TYPE "POWDER FEEDER HMI ACTIONS"
// stored: IsFailsafeCompliant false
   STRUCT
      SWITCH_ON_HEATER_LINE_1 : Bool;   // SWITCH ON HEATER LINE 1 HMI REQUEST
      SWITCH_OFF_HEATER_LINE_1 : Bool;   // SWITCH OFF HEATER LINE 1 HMI REQUEST
      SWITCHED_ON_HEATER_LINE_1 : Bool;   // SWITCHED ON HEATER LINE 1 HMI STATUS
      SWITCHED_OFF_HEATER_LINE_1 : Bool;   // SWITCHED OFF HEATER LINE 1 HMI STATUS
      SWITCH_ON_HEATER_LINE_2 : Bool;   // SWITCH ON HEATER LINE 2 HMI REQUEST
      SWITCH_OFF_HEATER_LINE_2 : Bool;   // SWITCH OFF HEATER LINE 2 HMI REQUEST
      SWITCHED_ON_HEATER_LINE_2 : Bool;   // SWITCHED ON HEATER LINE 2 HMI STATUS
      SWITCHED_OFF_HEATER_LINE_2 : Bool;   // SWITCHED OFF HEATER LINE 2 HMI STATUS
      SWITCH_ON_HOOPER_LINE_1 : Bool;   // SWITCH ON HOOPER LINE 1 HMI REQUEST
      SWITCH_OFF_HOOPER_LINE_1 : Bool;   // SWITCH OFF HOOPER LINE 1 HMI REQUEST
      SWITCHED_ON_HOOPER_LINE_1 : Bool;   // SWITCHED ON HOOPER LINE 1 HMI STATUS
      SWITCHED_OFF_HOOPER_LINE_1 : Bool;   // SWITCHED OFF HOOPER LINE 1 HMI STATUS
      SWITCH_ON_HOOPER_LINE_2 : Bool;   // SWITCH ON HOOPER LINE 2 HMI REQUEST
      SWITCH_OFF_HOOPER_LINE_2 : Bool;   // SWITCH OFF HOOPER LINE 2 HMI REQUEST
      SWITCHED_ON_HOOPER_LINE_2 : Bool;   // SWITCHED ON HOOPER LINE 2 HMI STATUS
      SWITCHED_OFF_HOOPER_LINE_2 : Bool;   // SWITCHED OFF HOOPER LINE 2 HMI STATUS
      SELECT_ARGON_GAS : Bool;   // SELECT ARGON GAS HMI REQUEST
      SELECT_NITROGEN_GAS : Bool;   // SELECT NITROGEN GAS HMI REQUEST
      SELECT_HELIUM_GAS : Bool;   // SELECT HELIUM GAS HMI REQUEST
      SELECT_ARGON30_GAS : Bool;   // SELECT ARGON30 GAS HMI REQUEST
      SELECTED_ARGON_GAS : Bool;   // SELECTED ARGON GAS HMI STATUS
      SELECTED_NITROGEN_GAS : Bool;   // SELECTED NITROGEN GAS HMI STATUS
      SELECTED_HELIUM_GAS : Bool;   // SELECTED HELIJM GAS HMI STATUS
      SELECTED_ARGON30_GAS : Bool;   // SELECTED ARGON30 GAS HMI STATUS
      SELECT_METRIC_UNITS : Bool;   // SELECT METRIC UNITS HMI REQUEST
      SELECT_IMPERIAL_UNITS : Bool;   // SELECT IMPERIAL UNITS HMI REQUEST
      SELECTED_METRIC_UNITS : Bool;   // SELECTED METRIC UNITS HMI STATUS
      SELECTED_IMPERIAL_UNITS : Bool;   // SELECTED IMPERIAL UNITS HMI STATUS
   END_STRUCT;
END_TYPE

TYPE "POWDER FEEDER HMI OFFSETS ALARMS WARNINGS"
// stored: IsFailsafeCompliant false
   STRUCT
      CarrierGasNominalLine1_Max_Alarm : Real;
      CarrierGasNominalLine2_Max_Alarm : Real;
      DiskSpeedNominalLine1_Max_Alarm : Real;
      DiskSpeedNominalLine2_Max_Alarm : Real;
      StirrerSpeedNominalLine1_Max_Alarm : Real;
      StirrerSpeedNominalLine2_Max_Alarm : Real;
      HopperTempNominalLine1_Max_Alarm : Real;
      HopperTempNominalLine2_Max_Alarm : Real;
      CarrierGasNominalLine1_Min_Alarm : Real;
      CarrierGasNominalLine2_Min_Alarm : Real;
      DiskSpeedNominalLine1_Min_Alarm : Real;
      DiskSpeedNominalLine2_Min_Alarm : Real;
      StirrerSpeedNominalLine1_Min_Alarm : Real;
      StirrerSpeedNominalLine2_Min_Alarm : Real;
      CarrierGasNominalLine1_Max_Warning : Real;
      CarrierGasNominalLine2_Max_Warning : Real;
      DiskSpeedNominalLine1_Max_Warning : Real;
      DiskSpeedNominalLine2_Max_Warning : Real;
      StirrerSpeedNominalLine1_Max_Warning : Real;
      StirrerSpeedNominalLine2_Max_Warning : Real;
      CarrierGasNominalLine1_Min_Warning : Real;
      CarrierGasNominalLine2_Min_Warning : Real;
      DiskSpeedNominalLine1_Min_Warning : Real;
      DiskSpeedNominalLine2_Min_Warning : Real;
      StirrerSpeedNominalLine1_Min_Warning : Real;
      StirrerSpeedNominalLine2_Min_Warning : Real;
      Spare26 : Real;
      Spare27 : Real;
      Spare28 : Real;
      Spare29 : Real;
      Spare30 : Real;
   END_STRUCT;
END_TYPE

TYPE "POWDER FEEDER HMI VALUES SETPOINTS"
// stored: IsFailsafeCompliant false
   STRUCT
      CarrierGasNominalLine1 : Real;
      CarrierGasNominalLine2 : Real;
      DiskSpeedNominalLine1 : Real;
      DiskSpeedNominalLine2 : Real;
      StirrerSpeedNominalLine1 : Real;
      StirrerSpeedNominalLine2 : Real;
      HopperTempNominalLine1 : Real;
      HopperTempNominalLine2 : Real;
      Spare8 : Real;
      Spare9 : Real;
      Spare10 : Real;
      Spare11 : Real;
      Spare12 : Real;
      Spare13 : Real;
      Spare14 : Real;
      Spare15 : Real;
   END_STRUCT;
END_TYPE

TYPE "POWDER FEEDER HOPPER"
// stored: IsFailsafeCompliant false
   STRUCT
      START_GENERAL_CONDITIONS : Bool;   // START GENERAL CONDITIONS
      START_INITIAL_CONDITIONS_LINE_1 : Bool;   // START INITIAL CONDITIONS LINE 1
      START_MANUAL_REQUEST_LINE_1 : Bool;   // START MANUAL REQUEST LINE 1
      START_INITIAL_CONDITIONS_LINE_2 : Bool;   // START INITIAL CONDITIONS LINE 2
      START_MANUAL_REQUEST_LINE_2 : Bool;   // START MANUAL REQUEST LINE 2
      START_AUTO_REQUEST : Bool;   // START AUTO REQUEST
      START_GLOBAL_REQUEST_LINE_1 : Bool;   // START GLOBAL REQUEST LINE 1
      START_COMMAND_LINE_1 : Bool;   // START COMMAND LINE 1
      START_LINE_1 : Bool;   // START LINE 1
      FEEDBACK_ON_LINE_1 : Bool;   // FEEDBACK ON LINE 1
      START_GLOBAL_REQUEST_LINE_2 : Bool;   // START GLOBAL REQUEST LINE 2
      START_COMMAND_LINE_2 : Bool;   // START COMMAND LINE 2
      START_LINE_2 : Bool;   // START LINE 2
      FEEDBACK_ON_LINE_2 : Bool;   // FEEDBACK ON LINE 2
      STOP_GENERAL_CONDITIONS : Bool;   // STOP GENERAL CONDITIONS
      STOP_INITIAL_CONDITIONS_LINE_1 : Bool;   // STOP INITIAL CONDITIONS LINE 1
      STOP_MANUAL_REQUEST_LINE_1 : Bool;   // STOP MANUAL REQUEST LINE 1
      STOP_INITIAL_CONDITIONS_LINE_2 : Bool;   // STOP INITIAL CONDITIONS LINE 2
      STOP_MANUAL_REQUEST_LINE_2 : Bool;   // STOP MANUAL REQUEST LINE 2
      STOP_AUTO_REQUEST : Bool;   // STOP AUTO REQUEST
      STOP_GLOBAL_REQUEST_LINE_1 : Bool;   // STOP GLOBAL REQUEST LINE 1
      STOP_COMMAND_LINE_1 : Bool;   // STOP COMMAND LINE 1
      STOP_LINE_1 : Bool;   // STOP LINE 1
      FEEDBACK_OFF_LINE_1 : Bool;   // FEEDBACK OFF LINE 1
      STOP_GLOBAL_REQUEST_LINE_2 : Bool;   // STOP GLOBAL REQUEST LINE 2
      STOP_COMMAND_LINE_2 : Bool;   // STOP COMMAND LINE 2
      STOP_LINE_2 : Bool;   // STOP LINE 2
      FEEDBACK_OFF_LINE_2 : Bool;   // FEEDBACK OFF LINE 2
      START_GENERAL_CONDITIONS_HELP : Bool;   // START GENERAL CONDITIONS HELP
      START_INITIAL_CONDITIONS_HELP : Bool;   // START INITIAL CONDITIONS HELP
      STOP_GENERAL_CONDITIONS_HELP : Bool;   // STOP GENERAL CONDITIONS HELP
      STOP_INITIAL_CONDITIONS_HELP : Bool;   // STOP INITIAL CONDITIONS HELP
      FAULT : Bool;   // FAULT
   END_STRUCT;
END_TYPE

TYPE "POWDER FEEDER PLC AUXILIAR"
// stored: IsFailsafeCompliant false
   STRUCT
      o_fCarrierGasSelect : Bool;   // 0 = Argon Selected, 1 = Nitrogen Selected / 1 = Argon, 2 = Nitrogen, 3 = Helium, 4 = Argon30
      o_fUnitSelect : Bool;   // 0 = Metric Units, 1 = SI
      i_fCarrierGasSelected_Line1 : Bool;   // 0 = Argon Selected, 1 = Nitrogen Selected / 1 = Argon, 2 = Nitrogen, 3 = Helium, 4 = Argon30
      i_fCarrierGasSelected_Line2 : Bool;   // 0 = Argon Selected, 1 = Nitrogen Selected / 1 = Argon, 2 = Nitrogen, 3 = Helium, 4 = Argon30
      i_fCarrierGasSelectedAux : Bool;   // 1 = Argon, 2 = Nitrogen, 3 = Helium, 4 = Argon30
      i_fUnitSelected_Line1 : Bool;   // 0 = Metric Units, 1 = SI / 0 = Metric System, 1 = Imperial
      i_fUnitSelected_Line2 : Bool;   // 0 = Metric Units, 1 = SI / 0 = Metric System, 1 = Imperial
      i_fUnitSelectedAux : Bool;   // 0 = Metric System, 1 = Imperial
      o_rCarriergasNominal_Line1 : Real;   // Carrier Gas Setpoint [NLPM] (0..16 NLPM)
      o_rCarriergasNominal_Line2 : Real;   // Carrier Gas Setpoint [NLPM] (0..16 NLPM)
      o_rDiskSpeedNominal_Line1 : Real;   // Disk Speed Setpoint [%] (0..100 %)
      o_rDiskSpeedNominal_Line2 : Real;   // Disk Speed Setpoint [%] (0..100 %)
      o_rStirrerSpeedNominal_Line1 : Real;   // Stirrer Speed Setpoint [%] (30 - 100%)
      o_rStirrerSpeedNominal_Line2 : Real;   // Stirrer Speed Setpoint [%] (30 - 100%)
      o_rHopperTempNominal_Line1 : Real;   // Hopper Temperature Setpoint [°C] (n/a for Twin 150 R1.0)
      o_rHopperTempNominal_Line2 : Real;   // Hopper Temperature Setpoint [°C] (n/a for Twin 150 R1.0)
      o_rLLlimitCarriergas_Line1 : Real;   // Carrier Gas Flow LL Limit [NLPM] (Absolute Value)
      o_rLLlimitCarriergas_Line2 : Real;   // Carrier Gas Flow LL Limit [NLPM] (Absolute Value)
      o_rLLlimitDiskSpeedNominal_Line1 : Real;   // Disk Speed LL Limit [%] (Absolute Value)
      o_rLLlimitDiskSpeedNominal_Line2 : Real;   // Disk Speed LL Limit [%] (Absolute Value)
      o_rLLlimitStirrerSpeedNominal_Line1 : Real;   // Stirrer Speed LL Limit [%] (Absolute Value)
      o_rLLlimitStirrerSpeedNominal_Line2 : Real;   // Stirrer Speed LL Limit [%] (Absolute Value)
      o_rLlimitCarriergas_Line1 : Real;   // Carrier Gas L Limit [NLPM] (Absolute Value)
      o_rLlimitCarriergas_Line2 : Real;   // Carrier Gas L Limit [NLPM] (Absolute Value)
      o_rLlimitDiskSpeedNominal_Line1 : Real;   // Disk Speed L Limit [%] (Absolute Value)
      o_rLlimitDiskSpeedNominal_Line2 : Real;   // Disk Speed L Limit [%] (Absolute Value)
      o_rLlimitStirrerSpeedNominal_Line1 : Real;   // Stirrer Speed L Limit [%] (Absolute Value)
      o_rLlimitStirrerSpeedNominal_Line2 : Real;   // Stirrer Speed L Limit [%] (Absolute Value)
      o_rHlimitCarriergas_Line1 : Real;   // Carrier Gas H Limit [NLPM] (Absolute Value)
      o_rHlimitCarriergas_Line2 : Real;   // Carrier Gas H Limit [NLPM] (Absolute Value)
      o_rHlimitDiskSpeedNominal_Line1 : Real;   // Disk Speed H Limit [%] (Absolute Value)
      o_rHlimitDiskSpeedNominal_Line2 : Real;   // Disk Speed H Limit [%] (Absolute Value)
      o_rHlimitStirrerSpeedNominal_Line1 : Real;   // Stirrer Speed H Limit [%] (Absolute Value)
      o_rHlimitStirrerSpeedNominal_Line2 : Real;   // Stirrer Speed H Limit [%] (Absolute Value)
      o_rHHlimitCarriergas_Line1 : Real;   // Carrier Gas HH Limit [NLPM] (Absolute Value)
      o_rHHlimitCarriergas_Line2 : Real;   // Carrier Gas HH Limit [NLPM] (Absolute Value)
      o_rHHlimitDiskSpeedNominal_Line1 : Real;   // Disk Speed HH Limit [%] (Absolute Value)
      o_rHHlimitDiskSpeedNominal_Line2 : Real;   // Disk Speed HH Limit [%] (Absolute Value)
      o_rHHlimitStirrerSpeedNominal_Line1 : Real;   // Stirrer Speed HH Limit [%] (Absolute Value)
      o_rHHlimitStirrerSpeedNominal_Line2 : Real;   // Stirrer Speed HH Limit [%] (Absolute Value)
      o_rHHlimitHopperTempNominal_Line1 : Real;   // Hopper Temperature HH Limit (ºC), (Absolute Value, N/a For Twin 150 R1.0)
      o_rHHlimitHopperTempNominal_Line2 : Real;   // Hopper Temperature HH Limit (ºC), (Absolute Value, N/a For Twin 150 R1.0)
      i_rCarriergasActual_Line1 : Real;   // Actual Value Carriergas Flow (NLPM)
      i_rCarriergasActual_Line2 : Real;   // Actual Value Carriergas Flow (NLPM)
      i_rDiskActual_Line1 : Real;   // Actual Value Disk Speed (%)
      i_rDiskActual_Line2 : Real;   // Actual Value Disk Speed (%)
      i_rStirrerActual_Line1 : Real;   // Actual Value Stirrer Speed (%)
      i_rStirrerActual_Line2 : Real;   // Actual Value Stirrer Speed (%)
      i_rFeedrateActual_Line1 : Real;   // N/A For Twin 150
      i_rFeedrateActual_Line2 : Real;   // N/A For Twin 150
      i_rHopperTempActual_Line1 : Real;   // Actual Value Hopper Temperature (ºC)
      i_rHopperTempActual_Line2 : Real;   // Actual Value Hopper Temperature (ºC)
      i_rHopperPressureActual_Line1 : Real;   // Actual Value Hopper Pressure (Bar)
      i_rHopperPressureActual_Line2 : Real;   // Actual Value Hopper Pressure (Bar)
   END_STRUCT;
END_TYPE

TYPE "POWDER SWITCH"
// stored: IsFailsafeCompliant false
   STRUCT
      "Hopper 1 General Conditions" : Bool;   // Hopper 1 General Conditions
      "Hopper 1 Initial Conditions" : Bool;   // Hopper 1 Initial Conditions
      "Hopper 1 Manual Request" : Bool;   // Hopper 1 Manual Request
      "Hopper 1 Auto Request" : Bool;   // Hopper 1 Auto Request
      "Hopper 1 Global Request" : Bool;   // Hopper 1 Global Request
      "Hopper 1 Command" : Bool;   // Hopper 1 Command
      "Hopper 1" : Bool;   // Hopper 1
      "Feedback Hopper 1" : Bool;   // Feedback Hopper 1
      "Hopper 2 General Conditions" : Bool;   // Hopper 2 General Conditions
      "Hopper 2 Initial Conditions" : Bool;   // Hopper 2 Initial Conditions
      "Hopper 2 Manual Request" : Bool;   // Hopper 2 Manual Request
      "Hopper 2 Auto Request" : Bool;   // Hopper 2 Auto Request
      "Hopper 2 Global Request" : Bool;   // Hopper 2 Global Request
      "Hopper 2 Command" : Bool;   // Hopper 2 Command
      "Hopper 2" : Bool;   // Hopper 2
      "Feedback Hopper 2" : Bool;   // Feedback Hopper 2
      "Hopper 1 General Conditions Help" : Bool;   // Hopper 1 General Conditions Help
      "Hopper 1 Initial Conditions Help" : Bool;   // Hopper 1 Initial Conditions Help
      "Hopper 2 General Conditions Help" : Bool;   // Hopper 2 General Conditions Help
      "Hopper 2 Initial Conditions Help" : Bool;   // Hopper 2 Initial Conditions Help
   END_STRUCT;
END_TYPE

TYPE "LBP_typeAlarmMsgs"
TITLE = PLC-Error / Messages / PLC errores/avisos / PLC-Fehler / Meldungen
// User data type for block LBP_AlarmMessage [DB2] / Tipo de dato de usuario para bloque LBP_AlarmMessage [DB2] / Anwender-Datentyp für Baustein LBP_AlarmMessage [DB2]
// stored: IsFailsafeCompliant false
   STRUCT
      Chan : Array[1..10] of Struct   // Von Kanal 1..10 / From Channel 1..10 / Desde el canal 1..10
         FDD : Array[0..15] of Bool;   // Vorschub deaktivieren / Feed disable / Desactivar avance
         RID : Array[0..15] of Bool;   // Einlesen deaktivieren / Read-in disable / Desactivar lectura
         NCSD : Array[0..15] of Bool;   // NC Start deaktivieren / NC start disable / Desactivar Marcha CN
         FdStop_1 : Array[0..15] of Bool;   // Vorschub-Stopp GEO-Achse 1 / Feed stop GEOaxis 1 / Parada del avance eje geométrico 1
         FdStop_2 : Array[0..15] of Bool;   // Vorschub-Stopp GEO-Achse 2 / Feed stop GEOaxis 2 / Parada del avance eje geométrico 2
         FdStop_3 : Array[0..15] of Bool;   // Vorschub-Stopp GEO-Achse 3 / Feed stop GEOaxis 3 / Parada del avance eje geométrico 3
      END_STRUCT;
      Axis : Array[1..31] of Struct   // Von Achse 1..31 / From Axis 1..31 / Desde el eje 1..31
         FdStop : Array[0..15] of Bool;   // Vorschub-Stopp Achse/Spindel / Feed stop axis/spindle / Parada del avance eje/cabezal
      END_STRUCT;
      AddValUserA0 : Array[0..63] of Int;   // Zusätzlicher Wert für Alarme im Anwenderbereich 0 (700000..700063) / Additional value for alarms in the user area 0 (700000..700063) / Valor adicional para alarmas en el área de usuario 0 (700000..700063)
      ChanA : Array[1..10] of Struct   // Von Kanal 1..10 / From Channel 1..10 / Desde el canal 1..10
         FDD_5C00xx : Array[0..15] of Bool;   // Vorschub deaktivieren Alarm Nr. 5C0000..5C0015 / Feed disable Alarm no. 5C0000..5C0015 / Desactivar avance n.º alarma 5C0000..5C0015
         FDD_RID_5C01xx : Array[0..31] of Bool;   // Vorschub und Einlesen deaktivieren Alarm Nr. 5C0100..5C0131 / Feed and read-in disable Alarm no. 5C0100..5C0131 / Desactivar avance y lectura n.º alarma 5C0100..5C0131
         RID_5C02xx : Array[0..31] of Bool;   // Einlesen deaktivieren Alarm Nr. 5C0200..5C0231 / Read-in disable Alarm no. 5C0200..5C0231 / Desactivar lectura n.º alarma 5C0200..5C0231
         NCSD_5C03xx : Array[0..15] of Bool;   // NC Start deaktivieren Alarm Nr. 5C0300..5C0315 / NC start disable Alarm no. 5C0300..5C0315 / Desactivar Marcha CN n.º alarma 5C0300..5C0315
         FdStop_1_5C11xx : Array[0..15] of Bool;   // Vorschub-Stopp GEO-Achse 1 Alarm Nr. 5C1100..5C1115 / Feed stop GEOaxis 1 Alarm no. 5C1100..5C1115 / Parada de avance eje geométrico 1 n.º alarma 5C1100..5C1115
         FdStop_2_5C12xx : Array[0..15] of Bool;   // Vorschub-Stopp GEO-Achse 2 Alarm Nr. 5C1200..5C1215 / Feed stop GEOaxis 2 Alarm no. 5C1200..5C1215 / Parada de avance eje geométrico 2 n.º alarma 5C1200..5C1215
         FdStop_3_5C13xx : Array[0..15] of Bool;   // Vorschub-Stopp GEO-Achse 3 Alarm Nr. 5C1300..5C1315 / Feed stop GEOaxis 3 Alarm no. 5C1300..5C1315 / Parada de avance eje geométrico 3 n.º alarma 5C1300..5C1315
      END_STRUCT;
      AxisA : Array[1..31] of Struct   // Von Achse 1..31 / From Axis 1..31 / Desde el eje 1..31
         AAFdStop60AAxx : Array[0..15] of Bool;   // Vorschub-Stopp Achse/Spindel / Feed stop axis/spindle / Parada del avance eje/cabezal
      END_STRUCT;
      res552 : Word;   // Reserviert / Reserved / Reservado
      UserA : Array[0..63] of Struct
         A70UUxx : Array[0..63] of Bool;   // Alarm 70UU00..70UU63 (Anwender-Bereich) / Alarm 70UU00..70UU63 (user area) / Alarma 70UU00..70UU63 (área de usuario)
      END_STRUCT;
   END_STRUCT;
   // // Chan[2].FDD : Vorschub deaktivieren / Feed disable / Desactivar avance
   // // Chan[3].FDD : Vorschub deaktivieren / Feed disable / Desactivar avance
   // // Chan[4].FDD : Vorschub deaktivieren / Feed disable / Desactivar avance
   // // Chan[5].FDD : Vorschub deaktivieren / Feed disable / Desactivar avance
   // // Chan[6].FDD : Vorschub deaktivieren / Feed disable / Desactivar avance
   // // Chan[7].FDD : Vorschub deaktivieren / Feed disable / Desactivar avance
   // // Chan[8].FDD : Vorschub deaktivieren / Feed disable / Desactivar avance
   // // Chan[9].FDD : Vorschub deaktivieren / Feed disable / Desactivar avance
   // // Chan[10].FDD : Vorschub deaktivieren / Feed disable / Desactivar avance
   // // Chan[2].RID : Einlesen deaktivieren / Read-in disable / Desactivar lectura
   // // Chan[3].RID : Einlesen deaktivieren / Read-in disable / Desactivar lectura
   // // Chan[4].RID : Einlesen deaktivieren / Read-in disable / Desactivar lectura
   // // Chan[5].RID : Einlesen deaktivieren / Read-in disable / Desactivar lectura
   // // Chan[6].RID : Einlesen deaktivieren / Read-in disable / Desactivar lectura
   // // Chan[7].RID : Einlesen deaktivieren / Read-in disable / Desactivar lectura
   // // Chan[8].RID : Einlesen deaktivieren / Read-in disable / Desactivar lectura
   // // Chan[9].RID : Einlesen deaktivieren / Read-in disable / Desactivar lectura
   // // Chan[10].RID : Einlesen deaktivieren / Read-in disable / Desactivar lectura
   // // Chan[2].NCSD : NC Start deaktivieren / NC start disable / Desactivar Marcha CN
   // // Chan[3].NCSD : NC Start deaktivieren / NC start disable / Desactivar Marcha CN
   // // Chan[4].NCSD : NC Start deaktivieren / NC start disable / Desactivar Marcha CN
   // // Chan[5].NCSD : NC Start deaktivieren / NC start disable / Desactivar Marcha CN
   // // Chan[6].NCSD : NC Start deaktivieren / NC start disable / Desactivar Marcha CN
   // // Chan[7].NCSD : NC Start deaktivieren / NC start disable / Desactivar Marcha CN
   // // Chan[8].NCSD : NC Start deaktivieren / NC start disable / Desactivar Marcha CN
   // // Chan[9].NCSD : NC Start deaktivieren / NC start disable / Desactivar Marcha CN
   // // Chan[10].NCSD : NC Start deaktivieren / NC start disable / Desactivar Marcha CN
   // // Chan[2].FdStop_1 : Vorschub-Stopp GEO-Achse 1 / Feed stop GEOaxis 1 / Parada del avance eje geométrico 1
   // // Chan[3].FdStop_1 : Vorschub-Stopp GEO-Achse 1 / Feed stop GEOaxis 1 / Parada del avance eje geométrico 1
   // // Chan[4].FdStop_1 : Vorschub-Stopp GEO-Achse 1 / Feed stop GEOaxis 1 / Parada del avance eje geométrico 1
   // // Chan[5].FdStop_1 : Vorschub-Stopp GEO-Achse 1 / Feed stop GEOaxis 1 / Parada del avance eje geométrico 1
   // // Chan[6].FdStop_1 : Vorschub-Stopp GEO-Achse 1 / Feed stop GEOaxis 1 / Parada del avance eje geométrico 1
   // // Chan[7].FdStop_1 : Vorschub-Stopp GEO-Achse 1 / Feed stop GEOaxis 1 / Parada del avance eje geométrico 1
   // // Chan[8].FdStop_1 : Vorschub-Stopp GEO-Achse 1 / Feed stop GEOaxis 1 / Parada del avance eje geométrico 1
   // // Chan[9].FdStop_1 : Vorschub-Stopp GEO-Achse 1 / Feed stop GEOaxis 1 / Parada del avance eje geométrico 1
   // // Chan[10].FdStop_1 : Vorschub-Stopp GEO-Achse 1 / Feed stop GEOaxis 1 / Parada del avance eje geométrico 1
   // // Chan[2].FdStop_2 : Vorschub-Stopp GEO-Achse 2 / Feed stop GEOaxis 2 / Parada del avance eje geométrico 2
   // // Chan[3].FdStop_2 : Vorschub-Stopp GEO-Achse 2 / Feed stop GEOaxis 2 / Parada del avance eje geométrico 2
   // // Chan[4].FdStop_2 : Vorschub-Stopp GEO-Achse 2 / Feed stop GEOaxis 2 / Parada del avance eje geométrico 2
   // // Chan[5].FdStop_2 : Vorschub-Stopp GEO-Achse 2 / Feed stop GEOaxis 2 / Parada del avance eje geométrico 2
   // // Chan[6].FdStop_2 : Vorschub-Stopp GEO-Achse 2 / Feed stop GEOaxis 2 / Parada del avance eje geométrico 2
   // // Chan[7].FdStop_2 : Vorschub-Stopp GEO-Achse 2 / Feed stop GEOaxis 2 / Parada del avance eje geométrico 2
   // // Chan[8].FdStop_2 : Vorschub-Stopp GEO-Achse 2 / Feed stop GEOaxis 2 / Parada del avance eje geométrico 2
   // // Chan[9].FdStop_2 : Vorschub-Stopp GEO-Achse 2 / Feed stop GEOaxis 2 / Parada del avance eje geométrico 2
   // // Chan[10].FdStop_2 : Vorschub-Stopp GEO-Achse 2 / Feed stop GEOaxis 2 / Parada del avance eje geométrico 2
   // // Chan[2].FdStop_3 : Vorschub-Stopp GEO-Achse 3 / Feed stop GEOaxis 3 / Parada del avance eje geométrico 3
   // // Chan[3].FdStop_3 : Vorschub-Stopp GEO-Achse 3 / Feed stop GEOaxis 3 / Parada del avance eje geométrico 3
   // // Chan[4].FdStop_3 : Vorschub-Stopp GEO-Achse 3 / Feed stop GEOaxis 3 / Parada del avance eje geométrico 3
   // // Chan[5].FdStop_3 : Vorschub-Stopp GEO-Achse 3 / Feed stop GEOaxis 3 / Parada del avance eje geométrico 3
   // // Chan[6].FdStop_3 : Vorschub-Stopp GEO-Achse 3 / Feed stop GEOaxis 3 / Parada del avance eje geométrico 3
   // // Chan[7].FdStop_3 : Vorschub-Stopp GEO-Achse 3 / Feed stop GEOaxis 3 / Parada del avance eje geométrico 3
   // // Chan[8].FdStop_3 : Vorschub-Stopp GEO-Achse 3 / Feed stop GEOaxis 3 / Parada del avance eje geométrico 3
   // // Chan[9].FdStop_3 : Vorschub-Stopp GEO-Achse 3 / Feed stop GEOaxis 3 / Parada del avance eje geométrico 3
   // // Chan[10].FdStop_3 : Vorschub-Stopp GEO-Achse 3 / Feed stop GEOaxis 3 / Parada del avance eje geométrico 3
   // // Chan[1] : Von Kanal 1..10 / From Channel 1..10 / Desde el canal 1..10
   // // Chan[2] : Von Kanal 1..10 / From Channel 1..10 / Desde el canal 1..10
   // // Chan[3] : Von Kanal 1..10 / From Channel 1..10 / Desde el canal 1..10
   // // Chan[4] : Von Kanal 1..10 / From Channel 1..10 / Desde el canal 1..10
   // // Chan[5] : Von Kanal 1..10 / From Channel 1..10 / Desde el canal 1..10
   // // Chan[6] : Von Kanal 1..10 / From Channel 1..10 / Desde el canal 1..10
   // // Chan[7] : Von Kanal 1..10 / From Channel 1..10 / Desde el canal 1..10
   // // Chan[8] : Von Kanal 1..10 / From Channel 1..10 / Desde el canal 1..10
   // // Chan[9] : Von Kanal 1..10 / From Channel 1..10 / Desde el canal 1..10
   // // Chan[10] : Von Kanal 1..10 / From Channel 1..10 / Desde el canal 1..10
   // // Axis[2].FdStop : Vorschub-Stopp Achse/Spindel / Feed stop axis/spindle / Parada del avance eje/cabezal
   // // Axis[3].FdStop : Vorschub-Stopp Achse/Spindel / Feed stop axis/spindle / Parada del avance eje/cabezal
   // // Axis[4].FdStop : Vorschub-Stopp Achse/Spindel / Feed stop axis/spindle / Parada del avance eje/cabezal
   // // Axis[5].FdStop : Vorschub-Stopp Achse/Spindel / Feed stop axis/spindle / Parada del avance eje/cabezal
   // // Axis[6].FdStop : Vorschub-Stopp Achse/Spindel / Feed stop axis/spindle / Parada del avance eje/cabezal
   // // Axis[7].FdStop : Vorschub-Stopp Achse/Spindel / Feed stop axis/spindle / Parada del avance eje/cabezal
   // // Axis[8].FdStop : Vorschub-Stopp Achse/Spindel / Feed stop axis/spindle / Parada del avance eje/cabezal
   // // Axis[9].FdStop : Vorschub-Stopp Achse/Spindel / Feed stop axis/spindle / Parada del avance eje/cabezal
   // // Axis[10].FdStop : Vorschub-Stopp Achse/Spindel / Feed stop axis/spindle / Parada del avance eje/cabezal
   // // Axis[11].FdStop : Vorschub-Stopp Achse/Spindel / Feed stop axis/spindle / Parada del avance eje/cabezal
   // // Axis[12].FdStop : Vorschub-Stopp Achse/Spindel / Feed stop axis/spindle / Parada del avance eje/cabezal
   // // Axis[13].FdStop : Vorschub-Stopp Achse/Spindel / Feed stop axis/spindle / Parada del avance eje/cabezal
   // // Axis[14].FdStop : Vorschub-Stopp Achse/Spindel / Feed stop axis/spindle / Parada del avance eje/cabezal
   // // Axis[15].FdStop : Vorschub-Stopp Achse/Spindel / Feed stop axis/spindle / Parada del avance eje/cabezal
   // // Axis[16].FdStop : Vorschub-Stopp Achse/Spindel / Feed stop axis/spindle / Parada del avance eje/cabezal
   // // Axis[17].FdStop : Vorschub-Stopp Achse/Spindel / Feed stop axis/spindle / Parada del avance eje/cabezal
   // // Axis[18].FdStop : Vorschub-Stopp Achse/Spindel / Feed stop axis/spindle / Parada del avance eje/cabezal
   // // Axis[19].FdStop : Vorschub-Stopp Achse/Spindel / Feed stop axis/spindle / Parada del avance eje/cabezal
   // // Axis[20].FdStop : Vorschub-Stopp Achse/Spindel / Feed stop axis/spindle / Parada del avance eje/cabezal
   // // Axis[21].FdStop : Vorschub-Stopp Achse/Spindel / Feed stop axis/spindle / Parada del avance eje/cabezal
   // // Axis[22].FdStop : Vorschub-Stopp Achse/Spindel / Feed stop axis/spindle / Parada del avance eje/cabezal
   // // Axis[23].FdStop : Vorschub-Stopp Achse/Spindel / Feed stop axis/spindle / Parada del avance eje/cabezal
   // // Axis[24].FdStop : Vorschub-Stopp Achse/Spindel / Feed stop axis/spindle / Parada del avance eje/cabezal
   // // Axis[25].FdStop : Vorschub-Stopp Achse/Spindel / Feed stop axis/spindle / Parada del avance eje/cabezal
   // // Axis[26].FdStop : Vorschub-Stopp Achse/Spindel / Feed stop axis/spindle / Parada del avance eje/cabezal
   // // Axis[27].FdStop : Vorschub-Stopp Achse/Spindel / Feed stop axis/spindle / Parada del avance eje/cabezal
   // // Axis[28].FdStop : Vorschub-Stopp Achse/Spindel / Feed stop axis/spindle / Parada del avance eje/cabezal
   // // Axis[29].FdStop : Vorschub-Stopp Achse/Spindel / Feed stop axis/spindle / Parada del avance eje/cabezal
   // // Axis[30].FdStop : Vorschub-Stopp Achse/Spindel / Feed stop axis/spindle / Parada del avance eje/cabezal
   // // Axis[31].FdStop : Vorschub-Stopp Achse/Spindel / Feed stop axis/spindle / Parada del avance eje/cabezal
   // // Axis[1] : Von Achse 1..31 / From Axis 1..31 / Desde el eje 1..31
   // // Axis[2] : Von Achse 1..31 / From Axis 1..31 / Desde el eje 1..31
   // // Axis[3] : Von Achse 1..31 / From Axis 1..31 / Desde el eje 1..31
   // // Axis[4] : Von Achse 1..31 / From Axis 1..31 / Desde el eje 1..31
   // // Axis[5] : Von Achse 1..31 / From Axis 1..31 / Desde el eje 1..31
   // // Axis[6] : Von Achse 1..31 / From Axis 1..31 / Desde el eje 1..31
   // // Axis[7] : Von Achse 1..31 / From Axis 1..31 / Desde el eje 1..31
   // // Axis[8] : Von Achse 1..31 / From Axis 1..31 / Desde el eje 1..31
   // // Axis[9] : Von Achse 1..31 / From Axis 1..31 / Desde el eje 1..31
   // // Axis[10] : Von Achse 1..31 / From Axis 1..31 / Desde el eje 1..31
   // // Axis[11] : Von Achse 1..31 / From Axis 1..31 / Desde el eje 1..31
   // // Axis[12] : Von Achse 1..31 / From Axis 1..31 / Desde el eje 1..31
   // // Axis[13] : Von Achse 1..31 / From Axis 1..31 / Desde el eje 1..31
   // // Axis[14] : Von Achse 1..31 / From Axis 1..31 / Desde el eje 1..31
   // // Axis[15] : Von Achse 1..31 / From Axis 1..31 / Desde el eje 1..31
   // // Axis[16] : Von Achse 1..31 / From Axis 1..31 / Desde el eje 1..31
   // // Axis[17] : Von Achse 1..31 / From Axis 1..31 / Desde el eje 1..31
   // // Axis[18] : Von Achse 1..31 / From Axis 1..31 / Desde el eje 1..31
   // // Axis[19] : Von Achse 1..31 / From Axis 1..31 / Desde el eje 1..31
   // // Axis[20] : Von Achse 1..31 / From Axis 1..31 / Desde el eje 1..31
   // // Axis[21] : Von Achse 1..31 / From Axis 1..31 / Desde el eje 1..31
   // // Axis[22] : Von Achse 1..31 / From Axis 1..31 / Desde el eje 1..31
   // // Axis[23] : Von Achse 1..31 / From Axis 1..31 / Desde el eje 1..31
   // // Axis[24] : Von Achse 1..31 / From Axis 1..31 / Desde el eje 1..31
   // // Axis[25] : Von Achse 1..31 / From Axis 1..31 / Desde el eje 1..31
   // // Axis[26] : Von Achse 1..31 / From Axis 1..31 / Desde el eje 1..31
   // // Axis[27] : Von Achse 1..31 / From Axis 1..31 / Desde el eje 1..31
   // // Axis[28] : Von Achse 1..31 / From Axis 1..31 / Desde el eje 1..31
   // // Axis[29] : Von Achse 1..31 / From Axis 1..31 / Desde el eje 1..31
   // // Axis[30] : Von Achse 1..31 / From Axis 1..31 / Desde el eje 1..31
   // // Axis[31] : Von Achse 1..31 / From Axis 1..31 / Desde el eje 1..31
   // // ChanA[2].FDD_5C00xx : Vorschub deaktivieren Alarm Nr. 5C0000..5C0015 / Feed disable Alarm no. 5C0000..5C0015 / Desactivar avance n.º alarma 5C0000..5C0015
   // // ChanA[3].FDD_5C00xx : Vorschub deaktivieren Alarm Nr. 5C0000..5C0015 / Feed disable Alarm no. 5C0000..5C0015 / Desactivar avance n.º alarma 5C0000..5C0015
   // // ChanA[4].FDD_5C00xx : Vorschub deaktivieren Alarm Nr. 5C0000..5C0015 / Feed disable Alarm no. 5C0000..5C0015 / Desactivar avance n.º alarma 5C0000..5C0015
   // // ChanA[5].FDD_5C00xx : Vorschub deaktivieren Alarm Nr. 5C0000..5C0015 / Feed disable Alarm no. 5C0000..5C0015 / Desactivar avance n.º alarma 5C0000..5C0015
   // // ChanA[6].FDD_5C00xx : Vorschub deaktivieren Alarm Nr. 5C0000..5C0015 / Feed disable Alarm no. 5C0000..5C0015 / Desactivar avance n.º alarma 5C0000..5C0015
   // // ChanA[7].FDD_5C00xx : Vorschub deaktivieren Alarm Nr. 5C0000..5C0015 / Feed disable Alarm no. 5C0000..5C0015 / Desactivar avance n.º alarma 5C0000..5C0015
   // // ChanA[8].FDD_5C00xx : Vorschub deaktivieren Alarm Nr. 5C0000..5C0015 / Feed disable Alarm no. 5C0000..5C0015 / Desactivar avance n.º alarma 5C0000..5C0015
   // // ChanA[9].FDD_5C00xx : Vorschub deaktivieren Alarm Nr. 5C0000..5C0015 / Feed disable Alarm no. 5C0000..5C0015 / Desactivar avance n.º alarma 5C0000..5C0015
   // // ChanA[10].FDD_5C00xx : Vorschub deaktivieren Alarm Nr. 5C0000..5C0015 / Feed disable Alarm no. 5C0000..5C0015 / Desactivar avance n.º alarma 5C0000..5C0015
   // // ChanA[2].FDD_RID_5C01xx : Vorschub und Einlesen deaktivieren Alarm Nr. 5C0100..5C0131 / Feed and read-in disable Alarm no. 5C0100..5C0131 / Desactivar avance y lectura n.º alarma 5C0100..5C0131
   // // ChanA[3].FDD_RID_5C01xx : Vorschub und Einlesen deaktivieren Alarm Nr. 5C0100..5C0131 / Feed and read-in disable Alarm no. 5C0100..5C0131 / Desactivar avance y lectura n.º alarma 5C0100..5C0131
   // // ChanA[4].FDD_RID_5C01xx : Vorschub und Einlesen deaktivieren Alarm Nr. 5C0100..5C0131 / Feed and read-in disable Alarm no. 5C0100..5C0131 / Desactivar avance y lectura n.º alarma 5C0100..5C0131
   // // ChanA[5].FDD_RID_5C01xx : Vorschub und Einlesen deaktivieren Alarm Nr. 5C0100..5C0131 / Feed and read-in disable Alarm no. 5C0100..5C0131 / Desactivar avance y lectura n.º alarma 5C0100..5C0131
   // // ChanA[6].FDD_RID_5C01xx : Vorschub und Einlesen deaktivieren Alarm Nr. 5C0100..5C0131 / Feed and read-in disable Alarm no. 5C0100..5C0131 / Desactivar avance y lectura n.º alarma 5C0100..5C0131
   // // ChanA[7].FDD_RID_5C01xx : Vorschub und Einlesen deaktivieren Alarm Nr. 5C0100..5C0131 / Feed and read-in disable Alarm no. 5C0100..5C0131 / Desactivar avance y lectura n.º alarma 5C0100..5C0131
   // // ChanA[8].FDD_RID_5C01xx : Vorschub und Einlesen deaktivieren Alarm Nr. 5C0100..5C0131 / Feed and read-in disable Alarm no. 5C0100..5C0131 / Desactivar avance y lectura n.º alarma 5C0100..5C0131
   // // ChanA[9].FDD_RID_5C01xx : Vorschub und Einlesen deaktivieren Alarm Nr. 5C0100..5C0131 / Feed and read-in disable Alarm no. 5C0100..5C0131 / Desactivar avance y lectura n.º alarma 5C0100..5C0131
   // // ChanA[10].FDD_RID_5C01xx : Vorschub und Einlesen deaktivieren Alarm Nr. 5C0100..5C0131 / Feed and read-in disable Alarm no. 5C0100..5C0131 / Desactivar avance y lectura n.º alarma 5C0100..5C0131
   // // ChanA[2].RID_5C02xx : Einlesen deaktivieren Alarm Nr. 5C0200..5C0231 / Read-in disable Alarm no. 5C0200..5C0231 / Desactivar lectura n.º alarma 5C0200..5C0231
   // // ChanA[3].RID_5C02xx : Einlesen deaktivieren Alarm Nr. 5C0200..5C0231 / Read-in disable Alarm no. 5C0200..5C0231 / Desactivar lectura n.º alarma 5C0200..5C0231
   // // ChanA[4].RID_5C02xx : Einlesen deaktivieren Alarm Nr. 5C0200..5C0231 / Read-in disable Alarm no. 5C0200..5C0231 / Desactivar lectura n.º alarma 5C0200..5C0231
   // // ChanA[5].RID_5C02xx : Einlesen deaktivieren Alarm Nr. 5C0200..5C0231 / Read-in disable Alarm no. 5C0200..5C0231 / Desactivar lectura n.º alarma 5C0200..5C0231
   // // ChanA[6].RID_5C02xx : Einlesen deaktivieren Alarm Nr. 5C0200..5C0231 / Read-in disable Alarm no. 5C0200..5C0231 / Desactivar lectura n.º alarma 5C0200..5C0231
   // // ChanA[7].RID_5C02xx : Einlesen deaktivieren Alarm Nr. 5C0200..5C0231 / Read-in disable Alarm no. 5C0200..5C0231 / Desactivar lectura n.º alarma 5C0200..5C0231
   // // ChanA[8].RID_5C02xx : Einlesen deaktivieren Alarm Nr. 5C0200..5C0231 / Read-in disable Alarm no. 5C0200..5C0231 / Desactivar lectura n.º alarma 5C0200..5C0231
   // // ChanA[9].RID_5C02xx : Einlesen deaktivieren Alarm Nr. 5C0200..5C0231 / Read-in disable Alarm no. 5C0200..5C0231 / Desactivar lectura n.º alarma 5C0200..5C0231
   // // ChanA[10].RID_5C02xx : Einlesen deaktivieren Alarm Nr. 5C0200..5C0231 / Read-in disable Alarm no. 5C0200..5C0231 / Desactivar lectura n.º alarma 5C0200..5C0231
   // // ChanA[2].NCSD_5C03xx : NC Start deaktivieren Alarm Nr. 5C0300..5C0315 / NC start disable Alarm no. 5C0300..5C0315 / Desactivar Marcha CN n.º alarma 5C0300..5C0315
   // // ChanA[3].NCSD_5C03xx : NC Start deaktivieren Alarm Nr. 5C0300..5C0315 / NC start disable Alarm no. 5C0300..5C0315 / Desactivar Marcha CN n.º alarma 5C0300..5C0315
   // // ChanA[4].NCSD_5C03xx : NC Start deaktivieren Alarm Nr. 5C0300..5C0315 / NC start disable Alarm no. 5C0300..5C0315 / Desactivar Marcha CN n.º alarma 5C0300..5C0315
   // // ChanA[5].NCSD_5C03xx : NC Start deaktivieren Alarm Nr. 5C0300..5C0315 / NC start disable Alarm no. 5C0300..5C0315 / Desactivar Marcha CN n.º alarma 5C0300..5C0315
   // // ChanA[6].NCSD_5C03xx : NC Start deaktivieren Alarm Nr. 5C0300..5C0315 / NC start disable Alarm no. 5C0300..5C0315 / Desactivar Marcha CN n.º alarma 5C0300..5C0315
   // // ChanA[7].NCSD_5C03xx : NC Start deaktivieren Alarm Nr. 5C0300..5C0315 / NC start disable Alarm no. 5C0300..5C0315 / Desactivar Marcha CN n.º alarma 5C0300..5C0315
   // // ChanA[8].NCSD_5C03xx : NC Start deaktivieren Alarm Nr. 5C0300..5C0315 / NC start disable Alarm no. 5C0300..5C0315 / Desactivar Marcha CN n.º alarma 5C0300..5C0315
   // // ChanA[9].NCSD_5C03xx : NC Start deaktivieren Alarm Nr. 5C0300..5C0315 / NC start disable Alarm no. 5C0300..5C0315 / Desactivar Marcha CN n.º alarma 5C0300..5C0315
   // // ChanA[10].NCSD_5C03xx : NC Start deaktivieren Alarm Nr. 5C0300..5C0315 / NC start disable Alarm no. 5C0300..5C0315 / Desactivar Marcha CN n.º alarma 5C0300..5C0315
   // // ChanA[2].FdStop_1_5C11xx : Vorschub-Stopp GEO-Achse 1 Alarm Nr. 5C1100..5C1115 / Feed stop GEOaxis 1 Alarm no. 5C1100..5C1115 / Parada de avance eje geométrico 1 n.º alarma 5C1100..5C1115
   // // ChanA[3].FdStop_1_5C11xx : Vorschub-Stopp GEO-Achse 1 Alarm Nr. 5C1100..5C1115 / Feed stop GEOaxis 1 Alarm no. 5C1100..5C1115 / Parada de avance eje geométrico 1 n.º alarma 5C1100..5C1115
   // // ChanA[4].FdStop_1_5C11xx : Vorschub-Stopp GEO-Achse 1 Alarm Nr. 5C1100..5C1115 / Feed stop GEOaxis 1 Alarm no. 5C1100..5C1115 / Parada de avance eje geométrico 1 n.º alarma 5C1100..5C1115
   // // ChanA[5].FdStop_1_5C11xx : Vorschub-Stopp GEO-Achse 1 Alarm Nr. 5C1100..5C1115 / Feed stop GEOaxis 1 Alarm no. 5C1100..5C1115 / Parada de avance eje geométrico 1 n.º alarma 5C1100..5C1115
   // // ChanA[6].FdStop_1_5C11xx : Vorschub-Stopp GEO-Achse 1 Alarm Nr. 5C1100..5C1115 / Feed stop GEOaxis 1 Alarm no. 5C1100..5C1115 / Parada de avance eje geométrico 1 n.º alarma 5C1100..5C1115
   // // ChanA[7].FdStop_1_5C11xx : Vorschub-Stopp GEO-Achse 1 Alarm Nr. 5C1100..5C1115 / Feed stop GEOaxis 1 Alarm no. 5C1100..5C1115 / Parada de avance eje geométrico 1 n.º alarma 5C1100..5C1115
   // // ChanA[8].FdStop_1_5C11xx : Vorschub-Stopp GEO-Achse 1 Alarm Nr. 5C1100..5C1115 / Feed stop GEOaxis 1 Alarm no. 5C1100..5C1115 / Parada de avance eje geométrico 1 n.º alarma 5C1100..5C1115
   // // ChanA[9].FdStop_1_5C11xx : Vorschub-Stopp GEO-Achse 1 Alarm Nr. 5C1100..5C1115 / Feed stop GEOaxis 1 Alarm no. 5C1100..5C1115 / Parada de avance eje geométrico 1 n.º alarma 5C1100..5C1115
   // // ChanA[10].FdStop_1_5C11xx : Vorschub-Stopp GEO-Achse 1 Alarm Nr. 5C1100..5C1115 / Feed stop GEOaxis 1 Alarm no. 5C1100..5C1115 / Parada de avance eje geométrico 1 n.º alarma 5C1100..5C1115
   // // ChanA[2].FdStop_2_5C12xx : Vorschub-Stopp GEO-Achse 2 Alarm Nr. 5C1200..5C1215 / Feed stop GEOaxis 2 Alarm no. 5C1200..5C1215 / Parada de avance eje geométrico 2 n.º alarma 5C1200..5C1215
   // // ChanA[3].FdStop_2_5C12xx : Vorschub-Stopp GEO-Achse 2 Alarm Nr. 5C1200..5C1215 / Feed stop GEOaxis 2 Alarm no. 5C1200..5C1215 / Parada de avance eje geométrico 2 n.º alarma 5C1200..5C1215
   // // ChanA[4].FdStop_2_5C12xx : Vorschub-Stopp GEO-Achse 2 Alarm Nr. 5C1200..5C1215 / Feed stop GEOaxis 2 Alarm no. 5C1200..5C1215 / Parada de avance eje geométrico 2 n.º alarma 5C1200..5C1215
   // // ChanA[5].FdStop_2_5C12xx : Vorschub-Stopp GEO-Achse 2 Alarm Nr. 5C1200..5C1215 / Feed stop GEOaxis 2 Alarm no. 5C1200..5C1215 / Parada de avance eje geométrico 2 n.º alarma 5C1200..5C1215
   // // ChanA[6].FdStop_2_5C12xx : Vorschub-Stopp GEO-Achse 2 Alarm Nr. 5C1200..5C1215 / Feed stop GEOaxis 2 Alarm no. 5C1200..5C1215 / Parada de avance eje geométrico 2 n.º alarma 5C1200..5C1215
   // // ChanA[7].FdStop_2_5C12xx : Vorschub-Stopp GEO-Achse 2 Alarm Nr. 5C1200..5C1215 / Feed stop GEOaxis 2 Alarm no. 5C1200..5C1215 / Parada de avance eje geométrico 2 n.º alarma 5C1200..5C1215
   // // ChanA[8].FdStop_2_5C12xx : Vorschub-Stopp GEO-Achse 2 Alarm Nr. 5C1200..5C1215 / Feed stop GEOaxis 2 Alarm no. 5C1200..5C1215 / Parada de avance eje geométrico 2 n.º alarma 5C1200..5C1215
   // // ChanA[9].FdStop_2_5C12xx : Vorschub-Stopp GEO-Achse 2 Alarm Nr. 5C1200..5C1215 / Feed stop GEOaxis 2 Alarm no. 5C1200..5C1215 / Parada de avance eje geométrico 2 n.º alarma 5C1200..5C1215
   // // ChanA[10].FdStop_2_5C12xx : Vorschub-Stopp GEO-Achse 2 Alarm Nr. 5C1200..5C1215 / Feed stop GEOaxis 2 Alarm no. 5C1200..5C1215 / Parada de avance eje geométrico 2 n.º alarma 5C1200..5C1215
   // // ChanA[2].FdStop_3_5C13xx : Vorschub-Stopp GEO-Achse 3 Alarm Nr. 5C1300..5C1315 / Feed stop GEOaxis 3 Alarm no. 5C1300..5C1315 / Parada de avance eje geométrico 3 n.º alarma 5C1300..5C1315
   // // ChanA[3].FdStop_3_5C13xx : Vorschub-Stopp GEO-Achse 3 Alarm Nr. 5C1300..5C1315 / Feed stop GEOaxis 3 Alarm no. 5C1300..5C1315 / Parada de avance eje geométrico 3 n.º alarma 5C1300..5C1315
   // // ChanA[4].FdStop_3_5C13xx : Vorschub-Stopp GEO-Achse 3 Alarm Nr. 5C1300..5C1315 / Feed stop GEOaxis 3 Alarm no. 5C1300..5C1315 / Parada de avance eje geométrico 3 n.º alarma 5C1300..5C1315
   // // ChanA[5].FdStop_3_5C13xx : Vorschub-Stopp GEO-Achse 3 Alarm Nr. 5C1300..5C1315 / Feed stop GEOaxis 3 Alarm no. 5C1300..5C1315 / Parada de avance eje geométrico 3 n.º alarma 5C1300..5C1315
   // // ChanA[6].FdStop_3_5C13xx : Vorschub-Stopp GEO-Achse 3 Alarm Nr. 5C1300..5C1315 / Feed stop GEOaxis 3 Alarm no. 5C1300..5C1315 / Parada de avance eje geométrico 3 n.º alarma 5C1300..5C1315
   // // ChanA[7].FdStop_3_5C13xx : Vorschub-Stopp GEO-Achse 3 Alarm Nr. 5C1300..5C1315 / Feed stop GEOaxis 3 Alarm no. 5C1300..5C1315 / Parada de avance eje geométrico 3 n.º alarma 5C1300..5C1315
   // // ChanA[8].FdStop_3_5C13xx : Vorschub-Stopp GEO-Achse 3 Alarm Nr. 5C1300..5C1315 / Feed stop GEOaxis 3 Alarm no. 5C1300..5C1315 / Parada de avance eje geométrico 3 n.º alarma 5C1300..5C1315
   // // ChanA[9].FdStop_3_5C13xx : Vorschub-Stopp GEO-Achse 3 Alarm Nr. 5C1300..5C1315 / Feed stop GEOaxis 3 Alarm no. 5C1300..5C1315 / Parada de avance eje geométrico 3 n.º alarma 5C1300..5C1315
   // // ChanA[10].FdStop_3_5C13xx : Vorschub-Stopp GEO-Achse 3 Alarm Nr. 5C1300..5C1315 / Feed stop GEOaxis 3 Alarm no. 5C1300..5C1315 / Parada de avance eje geométrico 3 n.º alarma 5C1300..5C1315
   // // ChanA[1] : Von Kanal 1..10 / From Channel 1..10 / Desde el canal 1..10
   // // ChanA[2] : Von Kanal 1..10 / From Channel 1..10 / Desde el canal 1..10
   // // ChanA[3] : Von Kanal 1..10 / From Channel 1..10 / Desde el canal 1..10
   // // ChanA[4] : Von Kanal 1..10 / From Channel 1..10 / Desde el canal 1..10
   // // ChanA[5] : Von Kanal 1..10 / From Channel 1..10 / Desde el canal 1..10
   // // ChanA[6] : Von Kanal 1..10 / From Channel 1..10 / Desde el canal 1..10
   // // ChanA[7] : Von Kanal 1..10 / From Channel 1..10 / Desde el canal 1..10
   // // ChanA[8] : Von Kanal 1..10 / From Channel 1..10 / Desde el canal 1..10
   // // ChanA[9] : Von Kanal 1..10 / From Channel 1..10 / Desde el canal 1..10
   // // ChanA[10] : Von Kanal 1..10 / From Channel 1..10 / Desde el canal 1..10
   // // AxisA[2].AAFdStop60AAxx : Vorschub-Stopp Achse/Spindel / Feed stop axis/spindle / Parada del avance eje/cabezal
   // // AxisA[3].AAFdStop60AAxx : Vorschub-Stopp Achse/Spindel / Feed stop axis/spindle / Parada del avance eje/cabezal
   // // AxisA[4].AAFdStop60AAxx : Vorschub-Stopp Achse/Spindel / Feed stop axis/spindle / Parada del avance eje/cabezal
   // // AxisA[5].AAFdStop60AAxx : Vorschub-Stopp Achse/Spindel / Feed stop axis/spindle / Parada del avance eje/cabezal
   // // AxisA[6].AAFdStop60AAxx : Vorschub-Stopp Achse/Spindel / Feed stop axis/spindle / Parada del avance eje/cabezal
   // // AxisA[7].AAFdStop60AAxx : Vorschub-Stopp Achse/Spindel / Feed stop axis/spindle / Parada del avance eje/cabezal
   // // AxisA[8].AAFdStop60AAxx : Vorschub-Stopp Achse/Spindel / Feed stop axis/spindle / Parada del avance eje/cabezal
   // // AxisA[9].AAFdStop60AAxx : Vorschub-Stopp Achse/Spindel / Feed stop axis/spindle / Parada del avance eje/cabezal
   // // AxisA[10].AAFdStop60AAxx : Vorschub-Stopp Achse/Spindel / Feed stop axis/spindle / Parada del avance eje/cabezal
   // // AxisA[11].AAFdStop60AAxx : Vorschub-Stopp Achse/Spindel / Feed stop axis/spindle / Parada del avance eje/cabezal
   // // AxisA[12].AAFdStop60AAxx : Vorschub-Stopp Achse/Spindel / Feed stop axis/spindle / Parada del avance eje/cabezal
   // // AxisA[13].AAFdStop60AAxx : Vorschub-Stopp Achse/Spindel / Feed stop axis/spindle / Parada del avance eje/cabezal
   // // AxisA[14].AAFdStop60AAxx : Vorschub-Stopp Achse/Spindel / Feed stop axis/spindle / Parada del avance eje/cabezal
   // // AxisA[15].AAFdStop60AAxx : Vorschub-Stopp Achse/Spindel / Feed stop axis/spindle / Parada del avance eje/cabezal
   // // AxisA[16].AAFdStop60AAxx : Vorschub-Stopp Achse/Spindel / Feed stop axis/spindle / Parada del avance eje/cabezal
   // // AxisA[17].AAFdStop60AAxx : Vorschub-Stopp Achse/Spindel / Feed stop axis/spindle / Parada del avance eje/cabezal
   // // AxisA[18].AAFdStop60AAxx : Vorschub-Stopp Achse/Spindel / Feed stop axis/spindle / Parada del avance eje/cabezal
   // // AxisA[19].AAFdStop60AAxx : Vorschub-Stopp Achse/Spindel / Feed stop axis/spindle / Parada del avance eje/cabezal
   // // AxisA[20].AAFdStop60AAxx : Vorschub-Stopp Achse/Spindel / Feed stop axis/spindle / Parada del avance eje/cabezal
   // // AxisA[21].AAFdStop60AAxx : Vorschub-Stopp Achse/Spindel / Feed stop axis/spindle / Parada del avance eje/cabezal
   // // AxisA[22].AAFdStop60AAxx : Vorschub-Stopp Achse/Spindel / Feed stop axis/spindle / Parada del avance eje/cabezal
   // // AxisA[23].AAFdStop60AAxx : Vorschub-Stopp Achse/Spindel / Feed stop axis/spindle / Parada del avance eje/cabezal
   // // AxisA[24].AAFdStop60AAxx : Vorschub-Stopp Achse/Spindel / Feed stop axis/spindle / Parada del avance eje/cabezal
   // // AxisA[25].AAFdStop60AAxx : Vorschub-Stopp Achse/Spindel / Feed stop axis/spindle / Parada del avance eje/cabezal
   // // AxisA[26].AAFdStop60AAxx : Vorschub-Stopp Achse/Spindel / Feed stop axis/spindle / Parada del avance eje/cabezal
   // // AxisA[27].AAFdStop60AAxx : Vorschub-Stopp Achse/Spindel / Feed stop axis/spindle / Parada del avance eje/cabezal
   // // AxisA[28].AAFdStop60AAxx : Vorschub-Stopp Achse/Spindel / Feed stop axis/spindle / Parada del avance eje/cabezal
   // // AxisA[29].AAFdStop60AAxx : Vorschub-Stopp Achse/Spindel / Feed stop axis/spindle / Parada del avance eje/cabezal
   // // AxisA[30].AAFdStop60AAxx : Vorschub-Stopp Achse/Spindel / Feed stop axis/spindle / Parada del avance eje/cabezal
   // // AxisA[31].AAFdStop60AAxx : Vorschub-Stopp Achse/Spindel / Feed stop axis/spindle / Parada del avance eje/cabezal
   // // AxisA[1] : Von Achse 1..31 / From Axis 1..31 / Desde el eje 1..31
   // // AxisA[2] : Von Achse 1..31 / From Axis 1..31 / Desde el eje 1..31
   // // AxisA[3] : Von Achse 1..31 / From Axis 1..31 / Desde el eje 1..31
   // // AxisA[4] : Von Achse 1..31 / From Axis 1..31 / Desde el eje 1..31
   // // AxisA[5] : Von Achse 1..31 / From Axis 1..31 / Desde el eje 1..31
   // // AxisA[6] : Von Achse 1..31 / From Axis 1..31 / Desde el eje 1..31
   // // AxisA[7] : Von Achse 1..31 / From Axis 1..31 / Desde el eje 1..31
   // // AxisA[8] : Von Achse 1..31 / From Axis 1..31 / Desde el eje 1..31
   // // AxisA[9] : Von Achse 1..31 / From Axis 1..31 / Desde el eje 1..31
   // // AxisA[10] : Von Achse 1..31 / From Axis 1..31 / Desde el eje 1..31
   // // AxisA[11] : Von Achse 1..31 / From Axis 1..31 / Desde el eje 1..31
   // // AxisA[12] : Von Achse 1..31 / From Axis 1..31 / Desde el eje 1..31
   // // AxisA[13] : Von Achse 1..31 / From Axis 1..31 / Desde el eje 1..31
   // // AxisA[14] : Von Achse 1..31 / From Axis 1..31 / Desde el eje 1..31
   // // AxisA[15] : Von Achse 1..31 / From Axis 1..31 / Desde el eje 1..31
   // // AxisA[16] : Von Achse 1..31 / From Axis 1..31 / Desde el eje 1..31
   // // AxisA[17] : Von Achse 1..31 / From Axis 1..31 / Desde el eje 1..31
   // // AxisA[18] : Von Achse 1..31 / From Axis 1..31 / Desde el eje 1..31
   // // AxisA[19] : Von Achse 1..31 / From Axis 1..31 / Desde el eje 1..31
   // // AxisA[20] : Von Achse 1..31 / From Axis 1..31 / Desde el eje 1..31
   // // AxisA[21] : Von Achse 1..31 / From Axis 1..31 / Desde el eje 1..31
   // // AxisA[22] : Von Achse 1..31 / From Axis 1..31 / Desde el eje 1..31
   // // AxisA[23] : Von Achse 1..31 / From Axis 1..31 / Desde el eje 1..31
   // // AxisA[24] : Von Achse 1..31 / From Axis 1..31 / Desde el eje 1..31
   // // AxisA[25] : Von Achse 1..31 / From Axis 1..31 / Desde el eje 1..31
   // // AxisA[26] : Von Achse 1..31 / From Axis 1..31 / Desde el eje 1..31
   // // AxisA[27] : Von Achse 1..31 / From Axis 1..31 / Desde el eje 1..31
   // // AxisA[28] : Von Achse 1..31 / From Axis 1..31 / Desde el eje 1..31
   // // AxisA[29] : Von Achse 1..31 / From Axis 1..31 / Desde el eje 1..31
   // // AxisA[30] : Von Achse 1..31 / From Axis 1..31 / Desde el eje 1..31
   // // AxisA[31] : Von Achse 1..31 / From Axis 1..31 / Desde el eje 1..31
   // // UserA[1].A70UUxx : Alarm 70UU00..70UU63 (Anwender-Bereich) / Alarm 70UU00..70UU63 (user area) / Alarma 70UU00..70UU63 (área de usuario)
   // // UserA[2].A70UUxx : Alarm 70UU00..70UU63 (Anwender-Bereich) / Alarm 70UU00..70UU63 (user area) / Alarma 70UU00..70UU63 (área de usuario)
   // // UserA[3].A70UUxx : Alarm 70UU00..70UU63 (Anwender-Bereich) / Alarm 70UU00..70UU63 (user area) / Alarma 70UU00..70UU63 (área de usuario)
   // // UserA[4].A70UUxx : Alarm 70UU00..70UU63 (Anwender-Bereich) / Alarm 70UU00..70UU63 (user area) / Alarma 70UU00..70UU63 (área de usuario)
   // // UserA[5].A70UUxx : Alarm 70UU00..70UU63 (Anwender-Bereich) / Alarm 70UU00..70UU63 (user area) / Alarma 70UU00..70UU63 (área de usuario)
   // // UserA[6].A70UUxx : Alarm 70UU00..70UU63 (Anwender-Bereich) / Alarm 70UU00..70UU63 (user area) / Alarma 70UU00..70UU63 (área de usuario)
   // // UserA[7].A70UUxx : Alarm 70UU00..70UU63 (Anwender-Bereich) / Alarm 70UU00..70UU63 (user area) / Alarma 70UU00..70UU63 (área de usuario)
   // // UserA[8].A70UUxx : Alarm 70UU00..70UU63 (Anwender-Bereich) / Alarm 70UU00..70UU63 (user area) / Alarma 70UU00..70UU63 (área de usuario)
   // // UserA[9].A70UUxx : Alarm 70UU00..70UU63 (Anwender-Bereich) / Alarm 70UU00..70UU63 (user area) / Alarma 70UU00..70UU63 (área de usuario)
   // // UserA[10].A70UUxx : Alarm 70UU00..70UU63 (Anwender-Bereich) / Alarm 70UU00..70UU63 (user area) / Alarma 70UU00..70UU63 (área de usuario)
   // // UserA[11].A70UUxx : Alarm 70UU00..70UU63 (Anwender-Bereich) / Alarm 70UU00..70UU63 (user area) / Alarma 70UU00..70UU63 (área de usuario)
   // // UserA[12].A70UUxx : Alarm 70UU00..70UU63 (Anwender-Bereich) / Alarm 70UU00..70UU63 (user area) / Alarma 70UU00..70UU63 (área de usuario)
   // // UserA[13].A70UUxx : Alarm 70UU00..70UU63 (Anwender-Bereich) / Alarm 70UU00..70UU63 (user area) / Alarma 70UU00..70UU63 (área de usuario)
   // // UserA[14].A70UUxx : Alarm 70UU00..70UU63 (Anwender-Bereich) / Alarm 70UU00..70UU63 (user area) / Alarma 70UU00..70UU63 (área de usuario)
   // // UserA[15].A70UUxx : Alarm 70UU00..70UU63 (Anwender-Bereich) / Alarm 70UU00..70UU63 (user area) / Alarma 70UU00..70UU63 (área de usuario)
   // // UserA[16].A70UUxx : Alarm 70UU00..70UU63 (Anwender-Bereich) / Alarm 70UU00..70UU63 (user area) / Alarma 70UU00..70UU63 (área de usuario)
   // // UserA[17].A70UUxx : Alarm 70UU00..70UU63 (Anwender-Bereich) / Alarm 70UU00..70UU63 (user area) / Alarma 70UU00..70UU63 (área de usuario)
   // // UserA[18].A70UUxx : Alarm 70UU00..70UU63 (Anwender-Bereich) / Alarm 70UU00..70UU63 (user area) / Alarma 70UU00..70UU63 (área de usuario)
   // // UserA[19].A70UUxx : Alarm 70UU00..70UU63 (Anwender-Bereich) / Alarm 70UU00..70UU63 (user area) / Alarma 70UU00..70UU63 (área de usuario)
   // // UserA[20].A70UUxx : Alarm 70UU00..70UU63 (Anwender-Bereich) / Alarm 70UU00..70UU63 (user area) / Alarma 70UU00..70UU63 (área de usuario)
   // // UserA[21].A70UUxx : Alarm 70UU00..70UU63 (Anwender-Bereich) / Alarm 70UU00..70UU63 (user area) / Alarma 70UU00..70UU63 (área de usuario)
   // // UserA[22].A70UUxx : Alarm 70UU00..70UU63 (Anwender-Bereich) / Alarm 70UU00..70UU63 (user area) / Alarma 70UU00..70UU63 (área de usuario)
   // // UserA[23].A70UUxx : Alarm 70UU00..70UU63 (Anwender-Bereich) / Alarm 70UU00..70UU63 (user area) / Alarma 70UU00..70UU63 (área de usuario)
   // // UserA[24].A70UUxx : Alarm 70UU00..70UU63 (Anwender-Bereich) / Alarm 70UU00..70UU63 (user area) / Alarma 70UU00..70UU63 (área de usuario)
   // // UserA[25].A70UUxx : Alarm 70UU00..70UU63 (Anwender-Bereich) / Alarm 70UU00..70UU63 (user area) / Alarma 70UU00..70UU63 (área de usuario)
   // // UserA[26].A70UUxx : Alarm 70UU00..70UU63 (Anwender-Bereich) / Alarm 70UU00..70UU63 (user area) / Alarma 70UU00..70UU63 (área de usuario)
   // // UserA[27].A70UUxx : Alarm 70UU00..70UU63 (Anwender-Bereich) / Alarm 70UU00..70UU63 (user area) / Alarma 70UU00..70UU63 (área de usuario)
   // // UserA[28].A70UUxx : Alarm 70UU00..70UU63 (Anwender-Bereich) / Alarm 70UU00..70UU63 (user area) / Alarma 70UU00..70UU63 (área de usuario)
   // // UserA[29].A70UUxx : Alarm 70UU00..70UU63 (Anwender-Bereich) / Alarm 70UU00..70UU63 (user area) / Alarma 70UU00..70UU63 (área de usuario)
   // // UserA[30].A70UUxx : Alarm 70UU00..70UU63 (Anwender-Bereich) / Alarm 70UU00..70UU63 (user area) / Alarma 70UU00..70UU63 (área de usuario)
   // // UserA[31].A70UUxx : Alarm 70UU00..70UU63 (Anwender-Bereich) / Alarm 70UU00..70UU63 (user area) / Alarma 70UU00..70UU63 (área de usuario)
   // // UserA[32].A70UUxx : Alarm 70UU00..70UU63 (Anwender-Bereich) / Alarm 70UU00..70UU63 (user area) / Alarma 70UU00..70UU63 (área de usuario)
   // // UserA[33].A70UUxx : Alarm 70UU00..70UU63 (Anwender-Bereich) / Alarm 70UU00..70UU63 (user area) / Alarma 70UU00..70UU63 (área de usuario)
   // // UserA[34].A70UUxx : Alarm 70UU00..70UU63 (Anwender-Bereich) / Alarm 70UU00..70UU63 (user area) / Alarma 70UU00..70UU63 (área de usuario)
   // // UserA[35].A70UUxx : Alarm 70UU00..70UU63 (Anwender-Bereich) / Alarm 70UU00..70UU63 (user area) / Alarma 70UU00..70UU63 (área de usuario)
   // // UserA[36].A70UUxx : Alarm 70UU00..70UU63 (Anwender-Bereich) / Alarm 70UU00..70UU63 (user area) / Alarma 70UU00..70UU63 (área de usuario)
   // // UserA[37].A70UUxx : Alarm 70UU00..70UU63 (Anwender-Bereich) / Alarm 70UU00..70UU63 (user area) / Alarma 70UU00..70UU63 (área de usuario)
   // // UserA[38].A70UUxx : Alarm 70UU00..70UU63 (Anwender-Bereich) / Alarm 70UU00..70UU63 (user area) / Alarma 70UU00..70UU63 (área de usuario)
   // // UserA[39].A70UUxx : Alarm 70UU00..70UU63 (Anwender-Bereich) / Alarm 70UU00..70UU63 (user area) / Alarma 70UU00..70UU63 (área de usuario)
   // // UserA[40].A70UUxx : Alarm 70UU00..70UU63 (Anwender-Bereich) / Alarm 70UU00..70UU63 (user area) / Alarma 70UU00..70UU63 (área de usuario)
   // // UserA[41].A70UUxx : Alarm 70UU00..70UU63 (Anwender-Bereich) / Alarm 70UU00..70UU63 (user area) / Alarma 70UU00..70UU63 (área de usuario)
   // // UserA[42].A70UUxx : Alarm 70UU00..70UU63 (Anwender-Bereich) / Alarm 70UU00..70UU63 (user area) / Alarma 70UU00..70UU63 (área de usuario)
   // // UserA[43].A70UUxx : Alarm 70UU00..70UU63 (Anwender-Bereich) / Alarm 70UU00..70UU63 (user area) / Alarma 70UU00..70UU63 (área de usuario)
   // // UserA[44].A70UUxx : Alarm 70UU00..70UU63 (Anwender-Bereich) / Alarm 70UU00..70UU63 (user area) / Alarma 70UU00..70UU63 (área de usuario)
   // // UserA[45].A70UUxx : Alarm 70UU00..70UU63 (Anwender-Bereich) / Alarm 70UU00..70UU63 (user area) / Alarma 70UU00..70UU63 (área de usuario)
   // // UserA[46].A70UUxx : Alarm 70UU00..70UU63 (Anwender-Bereich) / Alarm 70UU00..70UU63 (user area) / Alarma 70UU00..70UU63 (área de usuario)
   // // UserA[47].A70UUxx : Alarm 70UU00..70UU63 (Anwender-Bereich) / Alarm 70UU00..70UU63 (user area) / Alarma 70UU00..70UU63 (área de usuario)
   // // UserA[48].A70UUxx : Alarm 70UU00..70UU63 (Anwender-Bereich) / Alarm 70UU00..70UU63 (user area) / Alarma 70UU00..70UU63 (área de usuario)
   // // UserA[49].A70UUxx : Alarm 70UU00..70UU63 (Anwender-Bereich) / Alarm 70UU00..70UU63 (user area) / Alarma 70UU00..70UU63 (área de usuario)
   // // UserA[50].A70UUxx : Alarm 70UU00..70UU63 (Anwender-Bereich) / Alarm 70UU00..70UU63 (user area) / Alarma 70UU00..70UU63 (área de usuario)
   // // UserA[51].A70UUxx : Alarm 70UU00..70UU63 (Anwender-Bereich) / Alarm 70UU00..70UU63 (user area) / Alarma 70UU00..70UU63 (área de usuario)
   // // UserA[52].A70UUxx : Alarm 70UU00..70UU63 (Anwender-Bereich) / Alarm 70UU00..70UU63 (user area) / Alarma 70UU00..70UU63 (área de usuario)
   // // UserA[53].A70UUxx : Alarm 70UU00..70UU63 (Anwender-Bereich) / Alarm 70UU00..70UU63 (user area) / Alarma 70UU00..70UU63 (área de usuario)
   // // UserA[54].A70UUxx : Alarm 70UU00..70UU63 (Anwender-Bereich) / Alarm 70UU00..70UU63 (user area) / Alarma 70UU00..70UU63 (área de usuario)
   // // UserA[55].A70UUxx : Alarm 70UU00..70UU63 (Anwender-Bereich) / Alarm 70UU00..70UU63 (user area) / Alarma 70UU00..70UU63 (área de usuario)
   // // UserA[56].A70UUxx : Alarm 70UU00..70UU63 (Anwender-Bereich) / Alarm 70UU00..70UU63 (user area) / Alarma 70UU00..70UU63 (área de usuario)
   // // UserA[57].A70UUxx : Alarm 70UU00..70UU63 (Anwender-Bereich) / Alarm 70UU00..70UU63 (user area) / Alarma 70UU00..70UU63 (área de usuario)
   // // UserA[58].A70UUxx : Alarm 70UU00..70UU63 (Anwender-Bereich) / Alarm 70UU00..70UU63 (user area) / Alarma 70UU00..70UU63 (área de usuario)
   // // UserA[59].A70UUxx : Alarm 70UU00..70UU63 (Anwender-Bereich) / Alarm 70UU00..70UU63 (user area) / Alarma 70UU00..70UU63 (área de usuario)
   // // UserA[60].A70UUxx : Alarm 70UU00..70UU63 (Anwender-Bereich) / Alarm 70UU00..70UU63 (user area) / Alarma 70UU00..70UU63 (área de usuario)
   // // UserA[61].A70UUxx : Alarm 70UU00..70UU63 (Anwender-Bereich) / Alarm 70UU00..70UU63 (user area) / Alarma 70UU00..70UU63 (área de usuario)
   // // UserA[62].A70UUxx : Alarm 70UU00..70UU63 (Anwender-Bereich) / Alarm 70UU00..70UU63 (user area) / Alarma 70UU00..70UU63 (área de usuario)
   // // UserA[63].A70UUxx : Alarm 70UU00..70UU63 (Anwender-Bereich) / Alarm 70UU00..70UU63 (user area) / Alarma 70UU00..70UU63 (área de usuario)
END_TYPE

